// TIA Portal V19 export
DATA_BLOCK "RollformingMng_PERS"   // DB151
{ DB_Accessible_From_OPC_UA := 'FALSE' }
// stored: DBAccessibleFromOPCUA false, MemoryReserve 100
   VAR RETAIN
      PersistentValues : "udt_RollformingMng_Pers";
   END_VAR
BEGIN
   PersistentValues.Data.MaterialPresence := TRUE;
   PersistentValues.Data.MaterialPresence_Entry := TRUE;
   PersistentValues.Data.MaterialPresence_BeforeMW := TRUE;
   PersistentValues.Data.MaterialPresence_AfterMW := TRUE;
   PersistentValues.Data.MatPresence_ConveyorEntry := TRUE;
   PersistentValues.Data.FinalCut_DoneGood := FALSE;
   PersistentValues.Data.FinalCut_DoneWrong := FALSE;
   PersistentValues.Data.FinalCut_MemTargetResult := FALSE;
   PersistentValues.Data.ProfileHead_Found := TRUE;
   PersistentValues.Data.HeadingDone := TRUE;
   PersistentValues.Data.OldPPrf_PrgNo := 207;
   PersistentValues.Data.ActTarget.Ready := FALSE;
   PersistentValues.Data.ActTarget.P_ID := 0;
   PersistentValues.Data.ActTarget.O_ID := 0;
   PersistentValues.Data.ActTarget.Beam_Code := 0;
   PersistentValues.Data.ActTarget.X_Start := 0.0;
   PersistentValues.Data.ActTarget.X_End := 0.0;
   PersistentValues.Data.ActTarget.TargetTolerance := 0.0;
   PersistentValues.Data.ActTarget.PartLength := 0.0;
   PersistentValues.Data.ActTarget.DrawHead := FALSE;
   PersistentValues.Data.ActTarget.MarkHead := FALSE;
   PersistentValues.Data.ActTarget.WeldPresence := FALSE;
   PersistentValues.Data.NextTarget.Ready := FALSE;
   PersistentValues.Data.NextTarget.P_ID := 0;
   PersistentValues.Data.NextTarget.O_ID := 0;
   PersistentValues.Data.NextTarget.Beam_Code := 0;
   PersistentValues.Data.NextTarget.X_Start := 0.0;
   PersistentValues.Data.NextTarget.X_End := 0.0;
   PersistentValues.Data.NextTarget.TargetTolerance := 0.0;
   PersistentValues.Data.NextTarget.PartLength := 0.0;
   PersistentValues.Data.NextTarget.DrawHead := FALSE;
   PersistentValues.Data.NextTarget.MarkHead := FALSE;
   PersistentValues.Data.NextTarget.WeldPresence := FALSE;
   PersistentValues.Data.FS.LastCut_Material_Position := 689022.396252609;
   PersistentValues.Data.FS.LastJob_Material_Position := 689022.396252609;
   PersistentValues.Data.FS.PrevCut_Material_Position := 686325.050689577;
   PersistentValues.Data.FS.PrevJob_Material_Position := 686325.050689577;
   PersistentValues.Data.CutLenght.CarriageMeasID := 1994;
   PersistentValues.Data.CutLenght.WheelMeasID := 1994;
   PersistentValues.Data.CutLenght.CarriageEncoder := 1082.884;
   PersistentValues.Data.CutLenght.WheelEncoder := 520687.14;
   PersistentValues.Data.CutLenght.LastCut_Material_Position := 689022.574372612;
   PersistentValues.Data.CutLenght.PrevCut_Material_Position := 686325.054558052;
   PersistentValues.Par.Override.ProductionRateOverride := 75.0;
   PersistentValues.Par.Override.ChangeRateStepPercentage := 25.0;
   PersistentValues.Par.Override.EarlyPieces_Qty := 2;
   PersistentValues.Par.Override.EarlyPieces_Percentage := 30.0;
   PersistentValues.Par.Override.Emptying_Percentage := 30.0;
   PersistentValues.Par.Override.ProdSlowDow_Percentage := 50.0;
   PersistentValues.Par.Override.WeldPieces_Qty := 2;
   PersistentValues.Par.Override.WeldSlowDow_Percentage := 30.0;
   PersistentValues.Par.Override.AccRollSlowDown_Percentage := 100.0;
   PersistentValues.Par.SemiAut.Enable := TRUE;
   PersistentValues.Par.SemiAut.Vel := 10000.0;
   PersistentValues.Par.SemiAut.Acc := 1000.0;
   PersistentValues.Par.SemiAut.Dec := 1000.0;
   PersistentValues.Par.SemiAut.Jerk := 10000.0;
   PersistentValues.Par.AutoHeadingDistance := 3510.0;
   PersistentValues.Par.ExtractionDistance := 650.0;
   PersistentValues.Par.AccRollsDistanceFromZero := 1734.0;
END_DATA_BLOCK
